//  no ILO-mode >> cmd manual off to all used groups and reset all flags
      U     "MAL1S005".SecAc.Sta1On.Inf08;
      FN    DB895.DBX 3692.0;
      S     DB895.DBX 3006.0; // (ManOff)
      R     DB895.DBX 3014.0;
      R     DB895.DBX 3018.1;
//  Gr-cmd manual OFF
//  RESET ADDITIONAL CMD`S
//
//
// copy state
NETWORK
TITLE =ASW_9999: Init Flag
// clear all flags explicde to find them back
      U     "MAL1S005".PCRead.Step.StPassive; // explicid, to find them back
      R     "MAL1S005Par".Par.FlagFunction_1.StepLoading;
      R     "MAL1S005Par".Par.FlagFunction_1.StepUnloading;
      R     "MAL1S005Par".Par.FlagFunction_1.StepCleaning;
      R     "MAL1S005Par".Par.FlagFunction_1.LoadingBreak;
      R     "MAL1S005Par".Par.FlagFunction_1.UnloadingBreak;
      R     "MAL1S005Par".Par.FlagFunction_1.CleaningBreak;
      R     "MAL1S005Par".Par.FlagFunction_1.FinishLoading;
      R     "MAL1S005Par".Par.FlagFunction_1.FinishUnloading;
      R     "MAL1S005Par".Par.FlagFunction_1.FinishCleaning;
      R     "MAL1S005Par".Par.FlagFunction_1.TurningMeasure;
      R     "MAL1S005Par".Par.FlagFunction_1.MeasureHightLevel;
      R     "MAL1S005Par".Par.FlagFunction_1.TurningZeroPoint;
      R     "MAL1S005Par".Par.FlagFunction_1.Runde_1;
      R     "MAL1S005Par".Par.FlagFunction_1.Runde_2;
      R     "MAL1S005Par".Par.FlagFunction_1.Runde_3;
      R     "MAL1S005Par".Par.FlagFunction_1.Runde_4;
      R     "MAL1S005Par".Par.FlagFunction_1.Runde_5;
      R     "MAL1S005Par".Par.FlagFunction_1.Runde_6;
      R     "MAL1S005Par".Par.FlagFunction_1.Beladung_beendet;
      R     "MAL1S005Par".Par.FlagFunction_1.Entladerunden_erreicht;
      R     "MAL1S005Par".Par.FlagFunction_1.Reinigungsrunden_erreich;
      R     "MAL1S005Par".Par.FlagFunction_1.TurningStart;
      R     "MAL1S005Par".Par.FlagFunction_1.TurningStop;
      R     "MAL1S005Par".Par.FlagFunction_1.TurningLeft;
      R     "MAL1S005Par".Par.FlagFunction_1.TurningRight;
      R     "MAL1S005Par".Par.FlagFunction_1.LoadFirstPartEnd;
      R     "MAL1S005Par".Par.FlagFunction_1.TurningWithSpraying;
      R     "MAL1S005Par".Par.FlagFunction_1.TurningWithoutSpraying;
      R     "MAL1S005Par".Par.FlagFunction_1.UnloadEnd;
      R     "MAL1S005Par".Par.FlagFunction_1.UnloadSecondPartEnd;
      R     "MAL1S005Par".Par.FlagFunction_1.UnloadFirstPart;
      R     "MAL1S005Par".Par.FlagFunction_1.UnloadSecondPart;
      R     "MAL1S005Par".Par.FlagProcess.ProcessActive;
      R     "MAL1S005Par".Par.FlagProcess.ProcessStartFP;
      R     "MAL1S005Par".Par.FlagProcess.ProcessStartScan;
      R     "MAL1S005Par".Par.FlagProcess.ProcessEnd;
      R     "MAL1S005Par".Par.FlagProcess.ProcessEndFP;
      R     "MAL1S005Par".Par.FlagProcess.ProcessEndScan;
      R     "MAL1S005Par".Par.FlagProcess.NewStep;
      R     "MAL1S005Par".Par.FlagProcess.ReleaseProcessStart;
      R     "MAL1S005Par".Par.FlagProcess.FillingConditionatedWate;
      R     "MAL1S005Par".Par.FlagProcess.FillingFreshWater;
      R     "MAL1S005Par".Par.FlagProcess.SprayDuringFilling;
      R     "MAL1S005Par".Par.FlagProcess.AeriationDuringWaterFill;
      R     "MAL1S005Par".Par.FlagProcess.AeriatDurWaterFillFinish;
      R     "MAL1S005Par".Par.FlagProcess.SteepWaterFilled;
      R     "MAL1S005Par".Par.FlagProcess.SteepWaterFilledBySensor;
      R     "MAL1S005Par".Par.FlagProcess.CleaningSurface;
      R     "MAL1S005Par".Par.FlagFunction_0.CleaningSurfaceFinished;
      R     "MAL1S005Par".Par.FlagProcess1.DrainWaterAfterCleanSurf;
      R     "MAL1S005Par".Par.FlagProcess.CleaningSurface;
      R     "MAL1S005Par".Par.FlagProcess1.WaterDrainedAfterClSurf;
      R     "MAL1S005Par".Par.FlagProcess1.NoAerationBySteepFull;
      R     "MAL1S005Par".Par.FlagProcess.RunningCyclicAeriation;
      R     "MAL1S005Par".Par.FlagProcess.DrainWater;
      R     "MAL1S005Par".Par.FlagProcess1.WaterFilledForCleanSurf;
      R     "MAL1S005Par".Par.FlagFunction_0.StoreAerDuringWaterFill;
      R     "MAL1S005Par".Par.FlagFunction_0.CleaningGestartet;
      R     "MAL1S005Par".Par.FlagProcess.CO2Exhaust;
      R     "MAL1S005Par".Par.FlagProcess.RunningCyclicAeriation;
//
      SPBN  en13;
      L     L#0;
      T     "MAL1S005Par".Par.ProcessValue.ActualCondWater;
      T     "MAL1S005Par".Par.ProcessValue.ActualFreshWater;
      T     "MAL1S005Par".Par.ProcessValue.SummaryWaterOverall; // Volume of water
      L     0;
      T     "MAL1S005Par".ActTimeStepProcess.SteptimeActHour;
      T     "MAL1S005Par".ActTimeStepProcess.SteptimeActMin;
      T     "MAL1S005Par".ActTimeStepProcess.SteptimeActMinOverall;
en13: NOP   0;

      UN    "MAL1S005Par".Par.FlagProcess.ProcessActive;
      R     "MAL1S005Par".Par.FlagProcess.RunningCyclicAeriation;
      R     "MAL1S005Par".Par.FlagProcess.AeriationActive; // active aeriation
      R     "MAL1S005Par".Par.FlagProcess1.AeriationIntermittActive; // Aeriation Active
      R     "MAL1S005Par".Par.FlagProcess1.CO2SuckStart; // CO2 Suck Run
      R     "MAL1S005Par".Par.FlagProcess1.CO2SuckActive; // CO2 Suck Active
      R     "MAL1S005Par".Par.FlagProcess1.CO2SuckPause; // CO2 Suck Pause
      R     "MAL1S005Par".Par.FlagProcess.RunningCyclicAeriation;
      R     "MAL1S005Par".Par.FlagFunction_0.AeriationHTubeSelected;
      SPBN  rbit;
      L     0;
      T     "MAL1S005Par".Par.ParIntProcess.ActualDelayAeriation; // used as actual remaining period
      T     "MAL1S005Par".Par.ParIntProcess.ActualPauseAeriation;
      T     "MAL1S005Par".Par.ParIntProcess.ActualTimeAeriation;
      T     "MAL1S005Par".Par.ParIntProcess.ActualDelayCO2Suck; // used as actual remaining period
      T     "MAL1S005Par".Par.ParIntProcess.ActualPauseCO2Suck;
      T     "MAL1S005Par".Par.ParIntProcess.ActualTimeCO2Suck;
      T     "MAL1S005Par".Par.ParIntMachine.Value42;
      T     "MAL1S005Par".Par.ParIntProcess.ActualTimeCirculation; // used as actual remaining period
rbit: NOP   0;

NETWORK
TITLE =Main0_End: Init flag

      SET   ;
      R     "MAL1S005".Gr.All.CmdNewSelection;
      R     "MAL1S005".ToASW.CmdNewBatch;
      R     "MAL1S005".ToASW.CmdModify;

NETWORK
TITLE =End of block

      BE    ;

END_FUNCTION

